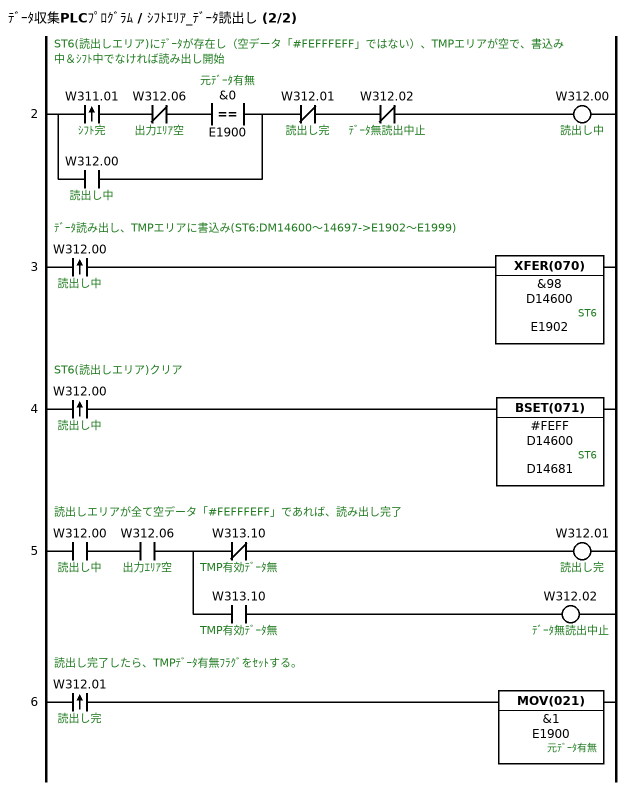
; [picture p24: ﾃﾞｰﾀ収集PLCﾌﾟﾛｸﾞﾗﾑ / ｼﾌﾄｴﾘｱ_ﾃﾞｰﾀ読出し, rungs 2-6]
; rung 2: ST6(読出しエリア)にﾃﾞｰﾀが存在し（空データ「#FEFFFEFF」ではない）、TMPエリアが空で、書込み中＆ｼﾌﾄ中でなければ読み出し開始
@LD W311.01  ; ｼﾌﾄ完
ANDNOT W312.06  ; 出力ｴﾘｱ空
AND=(300) &0 E1900  ; 元ﾃﾞｰﾀ有無
OR W312.00  ; 読出し中
ANDNOT W312.01  ; 読出し完
ANDNOT W312.02  ; ﾃﾞｰﾀ無読出中止
OUT W312.00  ; 読出し中
; rung 3: ﾃﾞｰﾀ読み出し、TMPエリアに書込み(ST6:DM14600～14697->E1902～E1999)
@LD W312.00  ; 読出し中
XFER(070) &98 D14600 E1902  ; ST6
; rung 4: ST6(読出しエリア)クリア
@LD W312.00  ; 読出し中
BSET(071) #FEFF D14600 D14681  ; ST6
; rung 5: 読出しエリアが全て空データ「#FEFFFEFF」であれば、読み出し完了
LD W312.00  ; 読出し中
AND W312.06  ; 出力ｴﾘｱ空
OUT TR0
ANDNOT W313.10  ; TMP有効ﾃﾞｰﾀ無
OUT W312.01  ; 読出し完
LD TR0
AND W313.10  ; TMP有効ﾃﾞｰﾀ無
OUT W312.02  ; ﾃﾞｰﾀ無読出中止
; rung 6: 読出し完了したら、TMPﾃﾞｰﾀ有無ﾌﾗｸﾞをｾｯﾄする。
@LD W312.01  ; 読出し完
MOV(021) &1 E1900  ; 元ﾃﾞｰﾀ有無

### Section ｼﾌﾄｴﾘｱ_ﾃﾞｰﾀｸﾘｱ

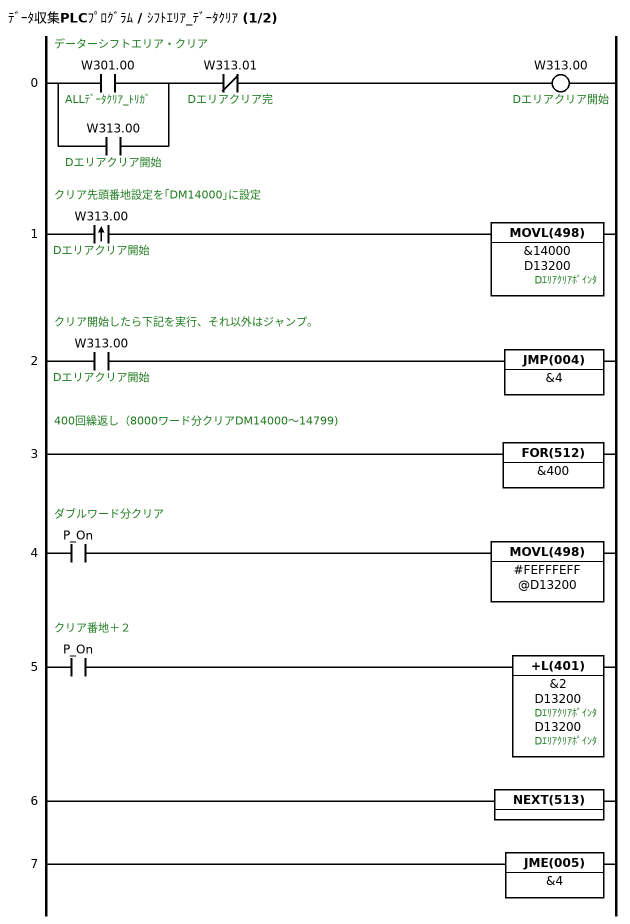
; rung 0: データーシフトエリア・クリア
LD W301.00  ; ALLﾃﾞｰﾀｸﾘｱ_ﾄﾘｶﾞ
OR W313.00  ; Dエリアクリア開始
ANDNOT W313.01  ; Dエリアクリア完
OUT W313.00  ; Dエリアクリア開始
; rung 1: クリア先頭番地設定を｢DM14000｣に設定
@LD W313.00  ; Dエリアクリア開始
MOVL(498) &14000 D13200  ; Dｴﾘｱｸﾘｱﾎﾟｲﾝﾀ
; rung 2: クリア開始したら下記を実行、それ以外はジャンプ。
LD W313.00  ; Dエリアクリア開始
JMP(004) &4
; rung 3: 400回繰返し（8000ワード分クリアDM14000～14799)
FOR(512) &400
; rung 4: ダブルワード分クリア
LD P_On
MOVL(498) #FEFFFEFF @D13200
; rung 5: クリア番地＋２
LD P_On
+L(401) &2 D13200 D13200  ; Dｴﾘｱｸﾘｱﾎﾟｲﾝﾀ
; rung 6
NEXT(513)
; rung 7
JME(005) &4

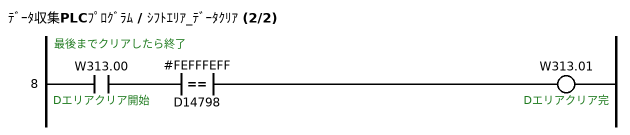
; rung 8: 最後までクリアしたら終了
LD W313.00  ; Dエリアクリア開始
AND=L(301) #FEFFFEFF D14798
OUT W313.01  ; Dエリアクリア完

### Section ｽﾀｯｸｴﾘｱ_ﾃﾞｰﾀ書込み

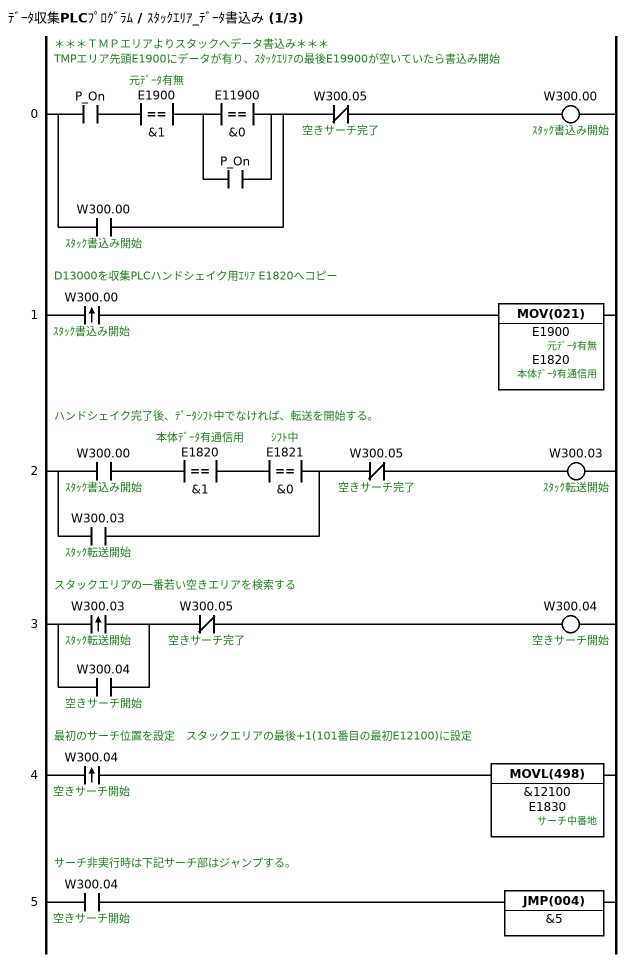
; rung 0: ＊＊＊ＴＭＰエリアよりスタックへデータ書込み＊＊＊ / TMPエリア先頭E1900にデータが有り、ｽﾀｯｸｴﾘｱの最後E19900が空いていたら書込み開始
LD P_On
AND=(300) E1900 &1  ; 元ﾃﾞｰﾀ有無
LD=(300) E11900 &0
OR P_On
ANDLD
OR W300.00  ; ｽﾀｯｸ書込み開始
ANDNOT W300.05  ; 空きサーチ完了
OUT W300.00  ; ｽﾀｯｸ書込み開始
; rung 1: D13000を収集PLCハンドシェイク用ｴﾘｱ E1820へコピー
@LD W300.00  ; ｽﾀｯｸ書込み開始
MOV(021) E1900 E1820  ; 元ﾃﾞｰﾀ有無, 本体ﾃﾞｰﾀ有通信用
; rung 2: ハンドシェイク完了後、ﾃﾞｰﾀｼﾌﾄ中でなければ、転送を開始する。
LD W300.00  ; ｽﾀｯｸ書込み開始
AND=(300) E1820 &1  ; 本体ﾃﾞｰﾀ有通信用
AND=(300) E1821 &0  ; ｼﾌﾄ中
OR W300.03  ; ｽﾀｯｸ転送開始
ANDNOT W300.05  ; 空きサーチ完了
OUT W300.03  ; ｽﾀｯｸ転送開始
; rung 3: スタックエリアの一番若い空きエリアを検索する
@LD W300.03  ; ｽﾀｯｸ転送開始
OR W300.04  ; 空きサーチ開始
ANDNOT W300.05  ; 空きサーチ完了
OUT W300.04  ; 空きサーチ開始
; rung 4: 最初のサーチ位置を設定　スタックエリアの最後+1(101番目の最初E12100)に設定
@LD W300.04  ; 空きサーチ開始
MOVL(498) &12100 E1830  ; サーチ中番地
; rung 5: サーチ非実行時は下記サーチ部はジャンプする。
LD W300.04  ; 空きサーチ開始
JMP(004) &5

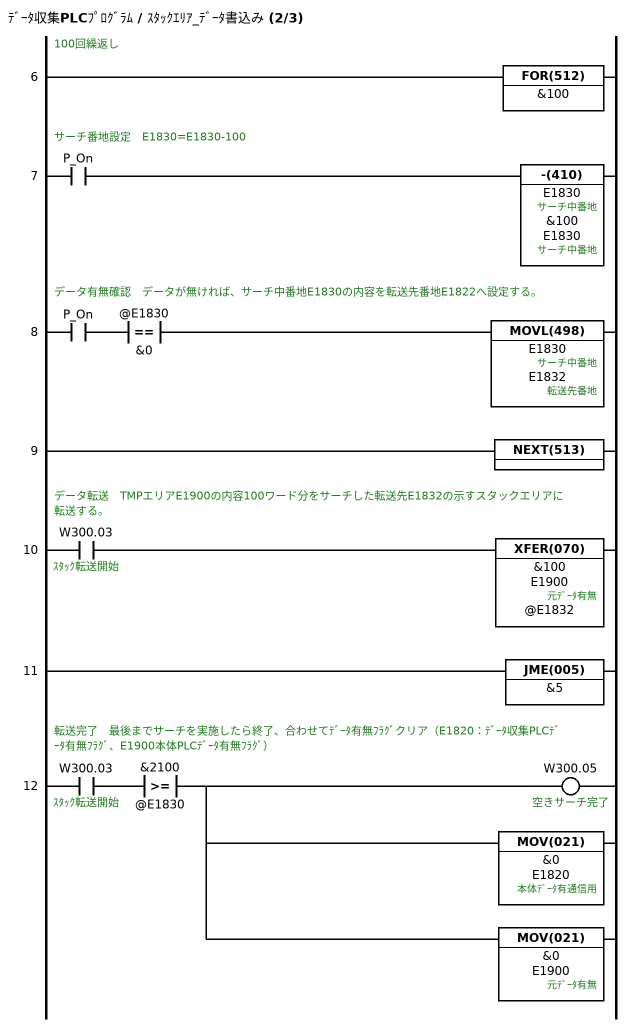
; rung 6: 100回繰返し
FOR(512) &100
; rung 7: サーチ番地設定　E1830=E1830-100
LD P_On
-(410) E1830 &100 E1830  ; サーチ中番地
; rung 8: データ有無確認　データが無ければ、サーチ中番地E1830の内容を転送先番地E1822へ設定する。
LD P_On
AND=(300) @E1830 &0
MOVL(498) E1830 E1832  ; サーチ中番地, 転送先番地
; rung 9
NEXT(513)
; rung 10: データ転送　TMPエリアE1900の内容100ワード分をサーチした転送先E1832の示すスタックエリアに転送する。
LD W300.03  ; ｽﾀｯｸ転送開始
XFER(070) &100 E1900 @E1832  ; 元ﾃﾞｰﾀ有無
; rung 11
JME(005) &5
; rung 12: 転送完了　最後までサーチを実施したら終了、合わせてﾃﾞｰﾀ有無ﾌﾗｸﾞクリア（E1820：ﾃﾞｰﾀ収集PLCﾃﾞｰﾀ有無ﾌﾗｸﾞ、E1900本体PLCﾃﾞｰﾀ有無ﾌﾗｸﾞ）
LD W300.03  ; ｽﾀｯｸ転送開始
AND>=(325) &2100 @E1830
OUT W300.05  ; 空きサーチ完了
MOV(021) &0 E1820  ; 本体ﾃﾞｰﾀ有通信用
MOV(021) &0 E1900  ; 元ﾃﾞｰﾀ有無

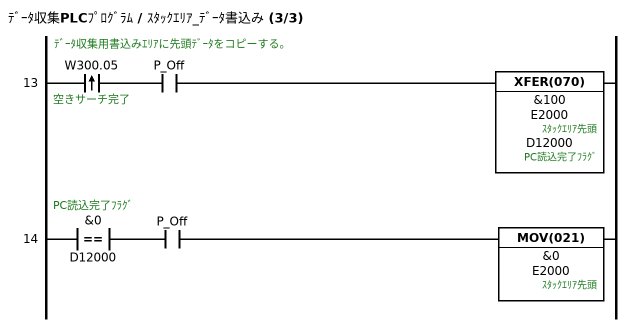
; rung 13: ﾃﾞｰﾀ収集用書込みｴﾘｱに先頭ﾃﾞｰﾀをコピーする。
@LD W300.05  ; 空きサーチ完了
AND P_Off
XFER(070) &100 E2000 D12000  ; ｽﾀｯｸｴﾘｱ先頭, PC読込完了ﾌﾗｸﾞ
; rung 14
LD=(300) &0 D12000  ; PC読込完了ﾌﾗｸﾞ
AND P_Off
MOV(021) &0 E2000  ; ｽﾀｯｸｴﾘｱ先頭

### Section ｽﾀｯｸｴﾘｱ_ﾃﾞｰﾀｼﾌﾄ

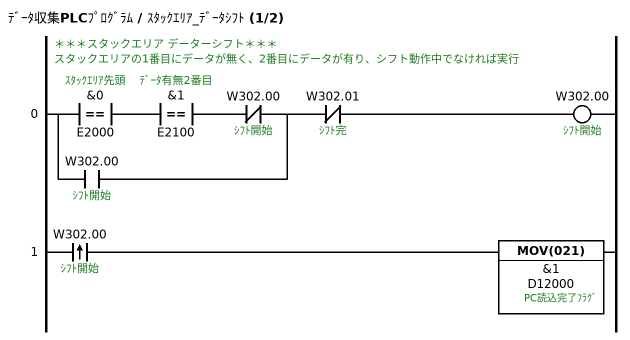
; rung 0: ＊＊＊スタックエリア データーシフト＊＊＊ / スタックエリアの1番目にデータが無く、2番目にデータが有り、シフト動作中でなければ実行
LD=(300) &0 E2000  ; ｽﾀｯｸｴﾘｱ先頭
AND=(300) &1 E2100  ; ﾃﾞｰﾀ有無2番目
ANDNOT W302.00  ; ｼﾌﾄ開始
OR W302.00  ; ｼﾌﾄ開始
ANDNOT W302.01  ; ｼﾌﾄ完
OUT W302.00  ; ｼﾌﾄ開始
; rung 1
@LD W302.00  ; ｼﾌﾄ開始
MOV(021) &1 D12000  ; PC読込完了ﾌﾗｸﾞ

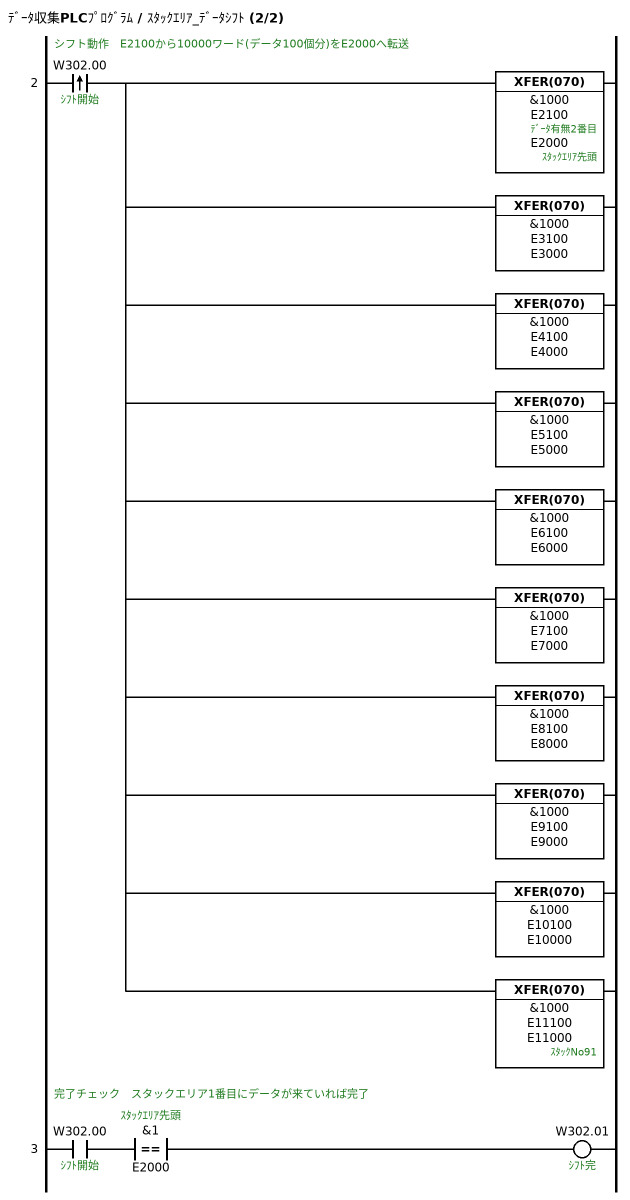
; rung 2: シフト動作　E2100から10000ワード(データ100個分)をE2000へ転送
@LD W302.00  ; ｼﾌﾄ開始
XFER(070) &1000 E2100 E2000  ; ﾃﾞｰﾀ有無2番目, ｽﾀｯｸｴﾘｱ先頭
XFER(070) &1000 E3100 E3000
XFER(070) &1000 E4100 E4000
XFER(070) &1000 E5100 E5000
XFER(070) &1000 E6100 E6000
XFER(070) &1000 E7100 E7000
XFER(070) &1000 E8100 E8000
XFER(070) &1000 E9100 E9000
XFER(070) &1000 E10100 E10000
XFER(070) &1000 E11100 E11000  ; ｽﾀｯｸNo91
; rung 3: 完了チェック　スタックエリア1番目にデータが来ていれば完了
LD W302.00  ; ｼﾌﾄ開始
AND=(300) &1 E2000  ; ｽﾀｯｸｴﾘｱ先頭
OUT W302.01  ; ｼﾌﾄ完

### Section ｽﾀｯｸｴﾘｱ_ﾃﾞｰﾀｸﾘｱ

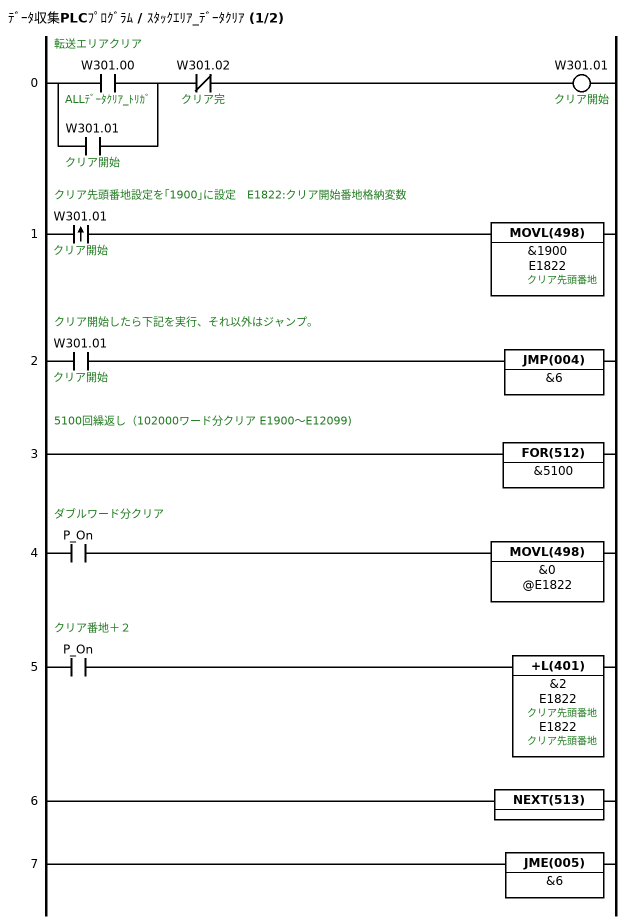
; rung 0: 転送エリアクリア
LD W301.00  ; ALLﾃﾞｰﾀｸﾘｱ_ﾄﾘｶﾞ
OR W301.01  ; クリア開始
ANDNOT W301.02  ; クリア完
OUT W301.01  ; クリア開始
; rung 1: クリア先頭番地設定を｢1900｣に設定　E1822:クリア開始番地格納変数
@LD W301.01  ; クリア開始
MOVL(498) &1900 E1822  ; クリア先頭番地
; rung 2: クリア開始したら下記を実行、それ以外はジャンプ。
LD W301.01  ; クリア開始
JMP(004) &6
; rung 3: 5100回繰返し（102000ワード分クリア E1900～E12099)
FOR(512) &5100
; rung 4: ダブルワード分クリア
LD P_On
MOVL(498) &0 @E1822
; rung 5: クリア番地＋２
LD P_On
+L(401) &2 E1822 E1822  ; クリア先頭番地
; rung 6
NEXT(513)
; rung 7
JME(005) &6

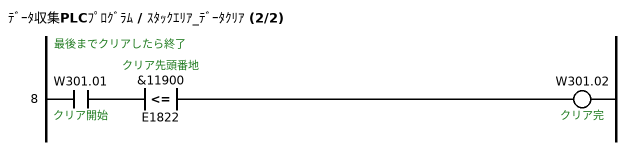
; rung 8: 最後までクリアしたら終了
LD W301.01  ; クリア開始
AND<=(315) &11900 E1822  ; クリア先頭番地
OUT W301.02  ; クリア完

### Section PCﾃﾞｰﾀ吸上げﾊﾝﾄﾞｼｪｲｸ

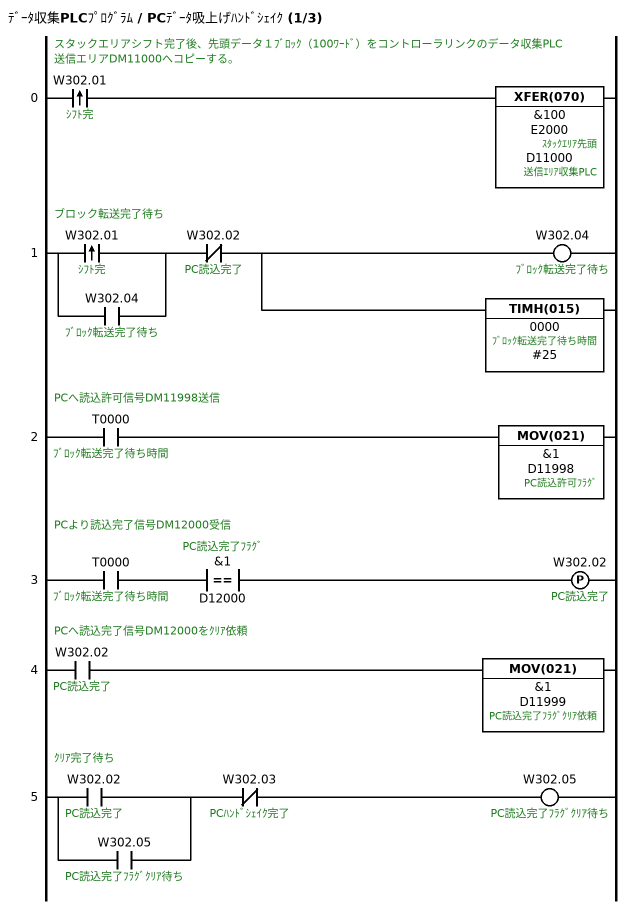
; rung 0: スタックエリアシフト完了後、先頭データ１ﾌﾞﾛｯｸ（100ﾜｰﾄﾞ）をコントローラリンクのデータ収集PLC送信エリアDM11000へコピーする。
@LD W302.01  ; ｼﾌﾄ完
XFER(070) &100 E2000 D11000  ; ｽﾀｯｸｴﾘｱ先頭, 送信ｴﾘｱ収集PLC
; rung 1: ブロック転送完了待ち
@LD W302.01  ; ｼﾌﾄ完
OR W302.04  ; ﾌﾞﾛｯｸ転送完了待ち
ANDNOT W302.02  ; PC読込完了
OUT W302.04  ; ﾌﾞﾛｯｸ転送完了待ち
TIMH(015) 0000 #25  ; ﾌﾞﾛｯｸ転送完了待ち時間
; rung 2: PCへ読込許可信号DM11998送信
LD T0000  ; ﾌﾞﾛｯｸ転送完了待ち時間
MOV(021) &1 D11998  ; PC読込許可ﾌﾗｸﾞ
; rung 3: PCより読込完了信号DM12000受信
LD T0000  ; ﾌﾞﾛｯｸ転送完了待ち時間
AND=(300) &1 D12000  ; PC読込完了ﾌﾗｸﾞ
DIFU(013) W302.02  ; PC読込完了
; rung 4: PCへ読込完了信号DM12000をｸﾘｱ依頼
LD W302.02  ; PC読込完了
MOV(021) &1 D11999  ; PC読込完了ﾌﾗｸﾞｸﾘｱ依頼
; rung 5: ｸﾘｱ完了待ち
LD W302.02  ; PC読込完了
OR W302.05  ; PC読込完了ﾌﾗｸﾞｸﾘｱ待ち
ANDNOT W302.03  ; PCﾊﾝﾄﾞｼｪｲｸ完了
OUT W302.05  ; PC読込完了ﾌﾗｸﾞｸﾘｱ待ち

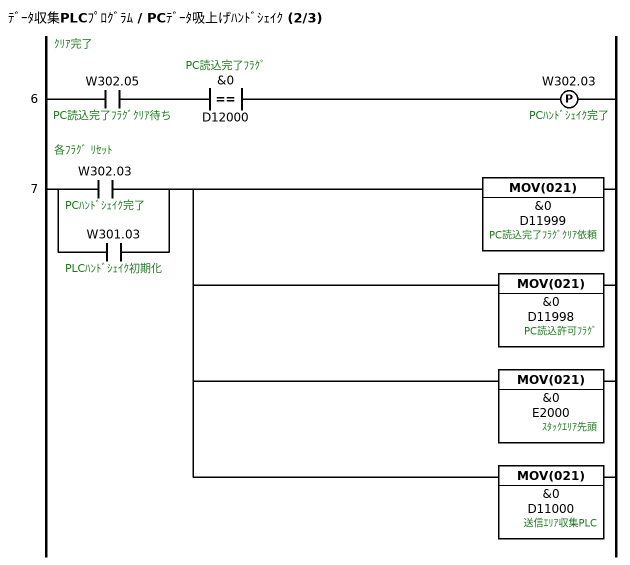
; rung 6: ｸﾘｱ完了
LD W302.05  ; PC読込完了ﾌﾗｸﾞｸﾘｱ待ち
AND=(300) &0 D12000  ; PC読込完了ﾌﾗｸﾞ
DIFU(013) W302.03  ; PCﾊﾝﾄﾞｼｪｲｸ完了
; rung 7: 各ﾌﾗｸﾞ ﾘｾｯﾄ
LD W302.03  ; PCﾊﾝﾄﾞｼｪｲｸ完了
OR W301.03  ; PLCﾊﾝﾄﾞｼｪｲｸ初期化
MOV(021) &0 D11999  ; PC読込完了ﾌﾗｸﾞｸﾘｱ依頼
MOV(021) &0 D11998  ; PC読込許可ﾌﾗｸﾞ
MOV(021) &0 E2000  ; ｽﾀｯｸｴﾘｱ先頭
MOV(021) &0 D11000  ; 送信ｴﾘｱ収集PLC

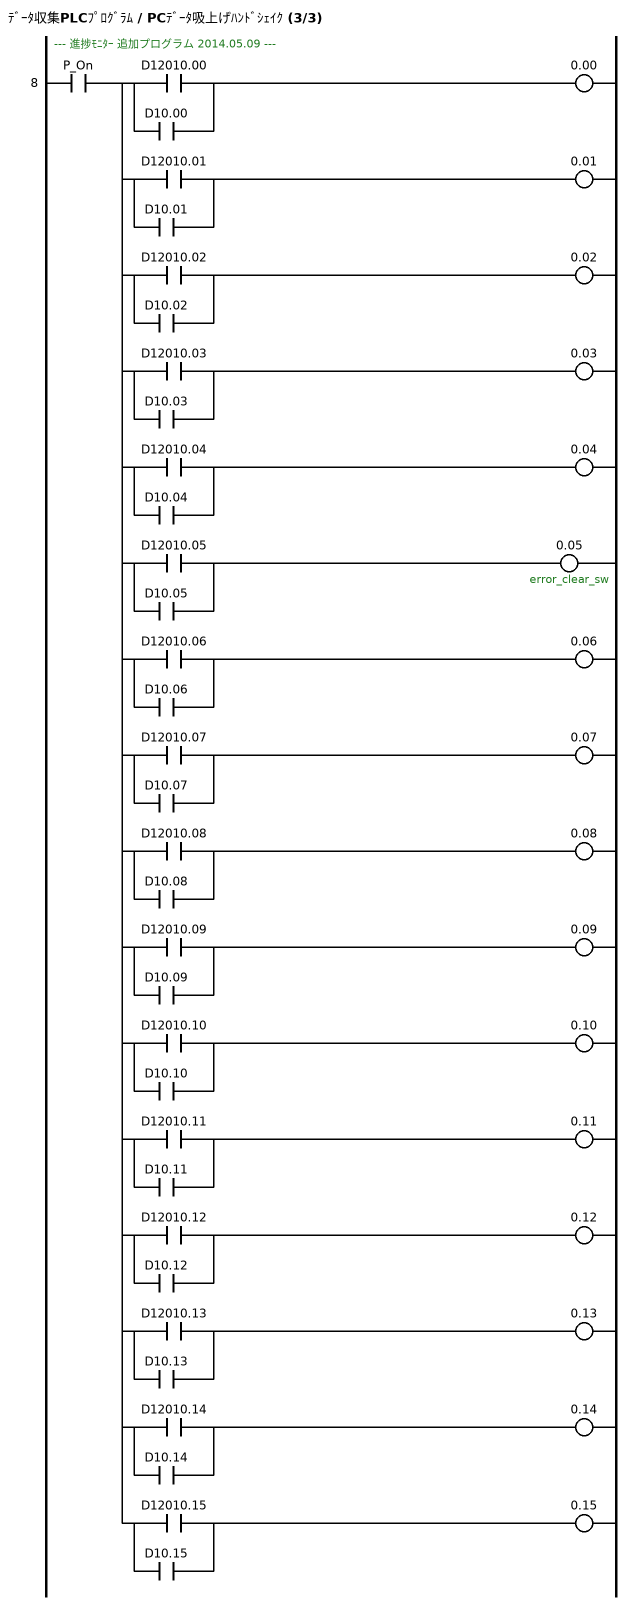
; rung 8: --- 進捗ﾓﾆﾀｰ 追加プログラム 2014.05.09 ---
LD P_On
OUT TR0
LD D12010.00
OR D10.00
ANDLD
OUT 0.00
LD TR0
LD D12010.01
OR D10.01
ANDLD
OUT 0.01
LD TR0
LD D12010.02
OR D10.02
ANDLD
OUT 0.02
LD TR0
LD D12010.03
OR D10.03
ANDLD
OUT 0.03
LD TR0
LD D12010.04
OR D10.04
ANDLD
OUT 0.04
LD TR0
LD D12010.05
OR D10.05
ANDLD
OUT 0.05  ; error_clear_sw
LD TR0
LD D12010.06
OR D10.06
ANDLD
OUT 0.06
LD TR0
LD D12010.07
OR D10.07
ANDLD
OUT 0.07
LD TR0
LD D12010.08
OR D10.08
ANDLD
OUT 0.08
LD TR0
LD D12010.09
OR D10.09
ANDLD
OUT 0.09
LD TR0
LD D12010.10
OR D10.10
ANDLD
OUT 0.10
LD TR0
LD D12010.11
OR D10.11
ANDLD
OUT 0.11
LD TR0
LD D12010.12
OR D10.12
ANDLD
OUT 0.12
LD TR0
LD D12010.13
OR D10.13
ANDLD
OUT 0.13
LD TR0
LD D12010.14
OR D10.14
ANDLD
OUT 0.14
LD TR0
LD D12010.15
OR D10.15
ANDLD
OUT 0.15

### Section END
; rung 0
END(001)